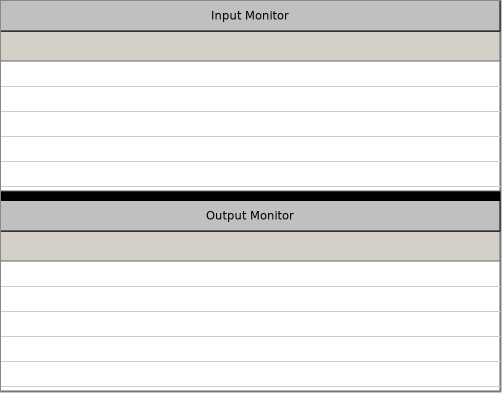
VISUALIZATION IO_Monitor  // 502x393
    Rectangle (0,0 500x391)
    Table (0,31 500x160), data array: InputByte
        p2232123230: Bit7
        p2685023577: InputByte[INDEX]
        p511219082: Bit6
        p1755163831: Bit5
        p4092479075: Bit4
        p2237128397: Bit3
        p505689113: Bit2
        p1757482276: Bit1
        p4088588272: Bit0
        Columns.Column.[3].Template: (InputByte[INDEX].4) <> 0; OnMouseDown: write the text variable via Edit
        Columns.Column.[4].Template: (InputByte[INDEX].3) <> 0; OnMouseDown: write the text variable via Edit
        Columns.Column.[5].Template: (InputByte[INDEX].2) <> 0; OnMouseDown: write the text variable via Edit
        Columns.Column.[0].Template: (InputByte[INDEX].7) <> 0; OnMouseDown: write the text variable via Edit
        Columns.Column.[1].Template: (InputByte[INDEX].6) <> 0; OnMouseDown: write the text variable via Edit
        Columns.Column.[6].Template: (InputByte[INDEX].1) <> 0; OnMouseDown: write the text variable via Edit
        Columns.Column.[2].Template: (InputByte[INDEX].5) <> 0; OnMouseDown: write the text variable via Edit
        Columns.Column.[7].Template: (InputByte[INDEX].0) <> 0; OnMouseDown: write the text variable via Edit
    Rectangle (0,0 500x31), "Input Monitor"
    Table (0,231 500x160), data array: OutputByte
        p2232123230: Bit7
        p511219082: Bit6
        p1755163831: Bit5
        p4092479075: Bit4
        p2237128397: Bit3
        p505689113: Bit2
        p1757482276: Bit1
        p4088588272: Bit0
        Columns.Column.[3].Template: (OutputByte[INDEX].4) <> 0; OnMouseDown: write the text variable via Edit
        Columns.Column.[4].Template: (OutputByte[INDEX].3) <> 0; OnMouseDown: write the text variable via Edit
        Columns.Column.[5].Template: (OutputByte[INDEX].2) <> 0; OnMouseDown: write the text variable via Edit
        Columns.Column.[0].Template: (OutputByte[INDEX].7) <> 0; OnMouseDown: write the text variable via Edit
        Columns.Column.[1].Template: (OutputByte[INDEX].6) <> 0; OnMouseDown: write the text variable via Edit
        Columns.Column.[6].Template: (OutputByte[INDEX].1) <> 0; OnMouseDown: write the text variable via Edit
        Columns.Column.[2].Template: (OutputByte[INDEX].5) <> 0; OnMouseDown: write the text variable via Edit
        Columns.Column.[7].Template: (OutputByte[INDEX].0) <> 0; OnMouseDown: write the text variable via Edit
    Rectangle (0,200 500x31), "Output Monitor"
END_VISUALIZATION

(* stored: Version 1.1.0.1, ProductVersion 3.1.4018.2
   Visu IO_Monitor: Id {6174a707-97bd-427c-825a-c8491fdeb8c4} *)
